// TIA Portal V17 export
// export: Created 2023-05-07T12:12:07.958498Z, ExportSetting WithDefaults, DisplayName Totally Integrated Automation Portal, DisplayVersion V17, DisplayName TIA Portal Openness, DisplayVersion V17, DisplayName TIA Portal Version Control Interface, DisplayVersion V17, DisplayName TIA Portal Test Suite Advanced, DisplayVersion V17, DisplayName STEP 7 Professional, DisplayVersion V17, DisplayName SIMATIC Energy Suite, DisplayVersion V17, DisplayName STEP 7 Safety, DisplayVersion V17, DisplayName WinCC Professional, DisplayVersion V17
FUNCTION "ControllerClass" : Void   // FC2, LAD
TITLE = ControllerClass
{ S7_Optimized_Access := 'TRUE' }
VERSION : 0.1
// stored: AutoNumber true, IsIECCheckEnabled false, SetENOAutomatically false, UDAEnableTagReadback false
   VAR_TEMP
      MV : Real;
      SP : Real;
   END_VAR
   VAR_TEMP   // added for the SCL form of the ladder/FBD networks
      _w1 : Bool;
   END_VAR
BEGIN

REGION Network 1: Call: Ramp
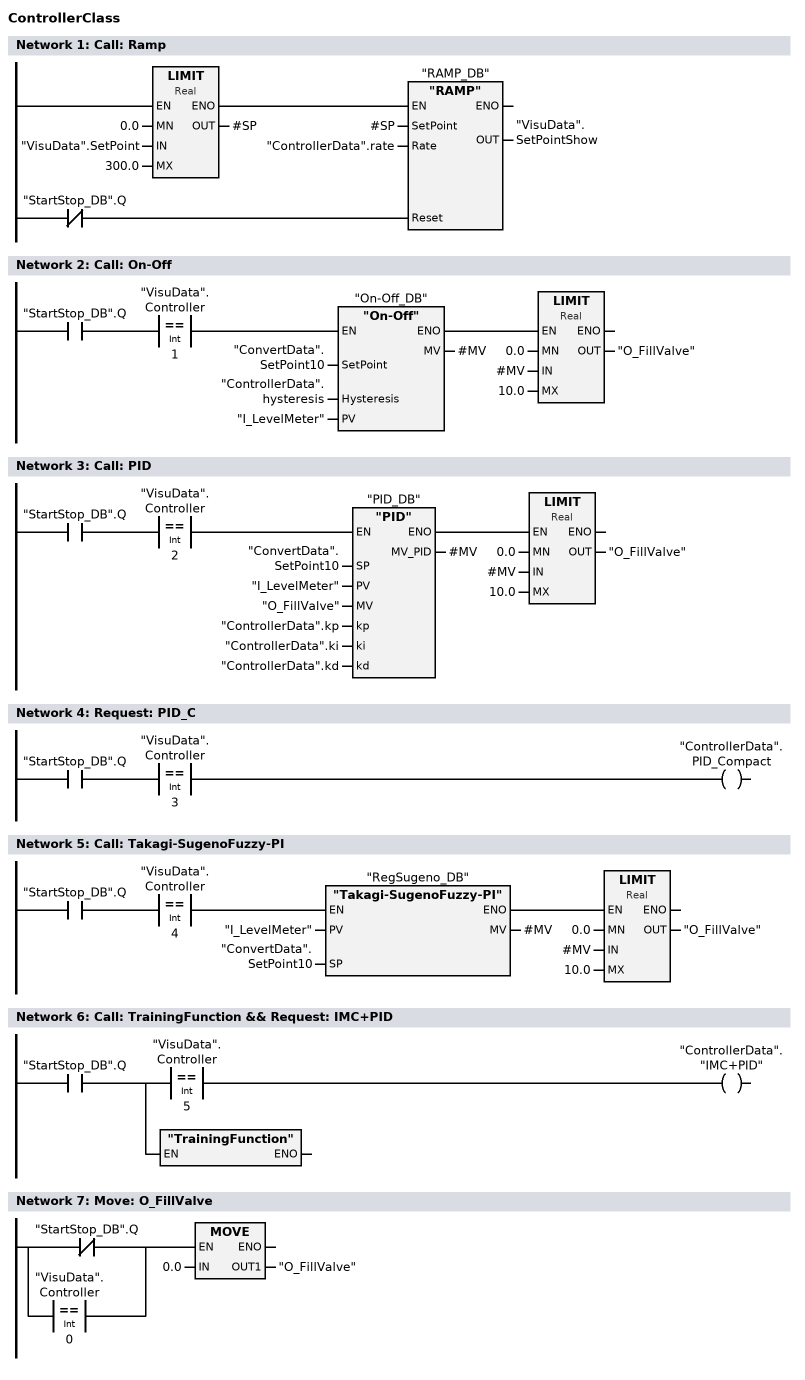
   RUNG wire#powerrail
      { S7_Templates := "value_type := Real" } Limit(mn := 0.0, in := "VisuData".SetPoint, mx := 300.0, out => #SP)
      "RAMP_DB"(Reset := wire#w1, SetPoint := #SP, Rate := "ControllerData".rate, OUT => "VisuData".SetPointShow)
   END_RUNG
   RUNG wire#powerrail
      I_Contact( "StartStop_DB".Q )
   END_RUNG wire#w1
   // the same network as SCL:
   #SP := LIMIT(MN := 0.0, IN := "VisuData".SetPoint, MX := 300.0);
   "RAMP_DB"(SetPoint := #SP,   // "RAMP"
             Rate := "ControllerData".rate,
             Reset := NOT "StartStop_DB".Q,
             OUT => "VisuData".SetPointShow);
END_REGION

REGION Network 2: Call: On-Off
   RUNG wire#powerrail
      Contact( "StartStop_DB".Q )
      { S7_Templates := "SrcType := Int" } EQ_Contact(in1 := "VisuData".Controller, in2 := 1)
      "On-Off_DB"(SetPoint := "ConvertData".SetPoint10, Hysteresis := "ControllerData".hysteresis, PV := "I_LevelMeter", MV => #MV)
      { S7_Templates := "value_type := Real" } Limit(mn := 0.0, in := #MV, mx := 10.0, out => "O_FillValve")
   END_RUNG
   // the same network as SCL:
   "On-Off_DB"(EN := "StartStop_DB".Q AND ("VisuData".Controller = 1),   // "On-Off"
               SetPoint := "ConvertData".SetPoint10,
               Hysteresis := "ControllerData".hysteresis,
               PV := "I_LevelMeter",
               MV => #MV,
               ENO => #_w1);
   IF #_w1 THEN "O_FillValve" := LIMIT(MN := 0.0, IN := #MV, MX := 10.0); END_IF;
END_REGION

REGION Network 3: Call: PID
   RUNG wire#powerrail
      Contact( "StartStop_DB".Q )
      { S7_Templates := "SrcType := Int" } EQ_Contact(in1 := "VisuData".Controller, in2 := 2)
      "PID_DB"(SP := "ConvertData".SetPoint10, PV := "I_LevelMeter", MV := "O_FillValve", kp := "ControllerData".kp, ki := "ControllerData".ki, kd := "ControllerData".kd, MV_PID => #MV)
      { S7_Templates := "value_type := Real" } Limit(mn := 0.0, in := #MV, mx := 10.0, out => "O_FillValve")
   END_RUNG
   // the same network as SCL:
   "PID_DB"(EN := "StartStop_DB".Q AND ("VisuData".Controller = 2),   // "PID"
            SP := "ConvertData".SetPoint10,
            PV := "I_LevelMeter",
            MV := "O_FillValve",
            kp := "ControllerData".kp,
            ki := "ControllerData".ki,
            kd := "ControllerData".kd,
            MV_PID => #MV,
            ENO => #_w1);
   IF #_w1 THEN "O_FillValve" := LIMIT(MN := 0.0, IN := #MV, MX := 10.0); END_IF;
END_REGION

REGION Network 4: Request: PID_C
   RUNG wire#powerrail
      Contact( "StartStop_DB".Q )
      { S7_Templates := "SrcType := Int" } EQ_Contact(in1 := "VisuData".Controller, in2 := 3)
      Coil( "ControllerData".PID_Compact )
   END_RUNG
   // the same network as SCL:
   "ControllerData".PID_Compact := "StartStop_DB".Q AND ("VisuData".Controller = 3);
END_REGION

REGION Network 5: Call: Takagi-SugenoFuzzy-PI
   RUNG wire#powerrail
      Contact( "StartStop_DB".Q )
      { S7_Templates := "SrcType := Int" } EQ_Contact(in1 := "VisuData".Controller, in2 := 4)
      "RegSugeno_DB"(PV := "I_LevelMeter", SP := "ConvertData".SetPoint10, MV => #MV)
      { S7_Templates := "value_type := Real" } Limit(mn := 0.0, in := #MV, mx := 10.0, out => "O_FillValve")
   END_RUNG
   // the same network as SCL:
   "RegSugeno_DB"(EN := "StartStop_DB".Q AND ("VisuData".Controller = 4),   // "Takagi-SugenoFuzzy-PI"
                  PV := "I_LevelMeter",
                  SP := "ConvertData".SetPoint10,
                  MV => #MV,
                  ENO => #_w1);
   IF #_w1 THEN "O_FillValve" := LIMIT(MN := 0.0, IN := #MV, MX := 10.0); END_IF;
END_REGION

REGION Network 6: Call: TrainingFunction && Request: IMC+PID
   RUNG wire#powerrail
      Contact( "StartStop_DB".Q )
      wire#w1
      { S7_Templates := "SrcType := Int" } EQ_Contact(in1 := "VisuData".Controller, in2 := 5)
      Coil( "ControllerData"."IMC+PID" )
   END_RUNG
   RUNG wire#w1
      "TrainingFunction"()
   END_RUNG
   // the same network as SCL:
   "ControllerData"."IMC+PID" := "StartStop_DB".Q AND ("VisuData".Controller = 5);
   IF "StartStop_DB".Q THEN "TrainingFunction"(); END_IF;
END_REGION

REGION Network 7: Move: O_FillValve
   RUNG wire#powerrail
      I_Contact( "StartStop_DB".Q )
      wire#w1
      Move(in := 0.0, out1 => "O_FillValve")
   END_RUNG
   RUNG wire#powerrail
      { S7_Templates := "SrcType := Int" } EQ_Contact(in1 := "VisuData".Controller, in2 := 0)
   END_RUNG wire#w1
   // the same network as SCL:
   IF NOT "StartStop_DB".Q OR ("VisuData".Controller = 0) THEN "O_FillValve" := 0.0; END_IF;
END_REGION
END_FUNCTION
